{attribute 'qualified_only'}
{attribute 'strict'}
TYPE eStates :
(
	INIT,
	START_EXECUTION,
	EXECUTING,
	DONE
);
END_TYPE

(* stored: Version 1.1.0.1, ProductVersion 3.1.4024.11
   DUT eStates: Id {ec67b23f-c2cf-474c-b72e-f502e60e4712} *)
